(*
SPDX-FileCopyrightText: © 2026 Oleksandr Tiutyk <trofimich@gmail.com>
SPDX-License-Identifier: MIT
License: https://opensource.org/license/mit
*)

(*!
<summary>Wrapper for native exception codes. The manager's static instance is a shared borrowed view.</summary>
<description>
Dynamic instances/clones belong to DynamicMemoryManager and must not be deleted manually.
Framework propagation preserves the captured code, catch point and timestamps in a dynamic clone.
</description>
*)

//!<param name="_AutoDisposeRegistrar">Dynamic system exceptions share the manager-owned lifetime of other exceptions.</param>

{attribute 'enable_dynamic_creation'}	
{attribute 'no_explicit_call' := 'do not call this function block directly'} 


FUNCTION_BLOCK SystemException EXTENDS Object IMPLEMENTS IException
VAR
	{attribute 'hide'} 
	_ClassName : STRING := __POUNAME();

	{attribute 'hide'} 
	_ExceptionCode : __SYSTEM.ExceptionCode;
	_LocalTimestamp : LDATE_AND_TIME;
	_UtcTimestamp : LDATE_AND_TIME;
	{attribute 'hide'} 	
	_CatchPointNamespaceName : STRING;
	{attribute 'hide'} 
	_CatchPointPOUName : STRING;
	{attribute 'hide'} 
	_CatchPointPosition : STRING;
	
	{attribute 'hide'} 
	_UnspecifiedPOU : STRING(128);

	{attribute 'hide'} 
	_UnspecifiedPosition : STRING(32);

	
	_AutoDisposeRegistrar : AutoDisposeRegistrar(THIS^);
END_VAR

METHOD PRIVATE appendTimestampDescription
VAR_IN_OUT CONSTANT
	stringBuilder : WideStringBuilder;
END_VAR
VAR_INPUT
	timestampDisplayMode : TIMESTAMP_DISPLAY_MODE := TIMESTAMP_DISPLAY_MODE.HIDDEN;
	localTimestamp : LDATE_AND_TIME;	
	utcTimestamp : LDATE_AND_TIME;	
END_VAR
IF timestampDisplayMode = TIMESTAMP_DISPLAY_MODE.HIDDEN THEN
	RETURN;
END_IF

CASE timestampDisplayMode OF
	TIMESTAMP_DISPLAY_MODE.LOCAL:
		stringBuilder.Append(localTimestamp);
	
	TIMESTAMP_DISPLAY_MODE.UTC:
		stringBuilder.Append(utcTimestamp).AppendString("UTC");
END_CASE
END_METHOD

{attribute 'monitoring' := 'call'}
PROPERTY ClassName : REFERENCE TO STRING
GET
ClassName REF= _ClassName;
END_GET
END_PROPERTY

(*!
<summary>Clears the code: Empty becomes TRUE and GetMessage returns an empty string.</summary>
<description>
Resets captured timestamps; does not delete/unregister the instance. Catch-point storage is retained.
</description>
*)

METHOD Clear
_ExceptionCode := __SYSTEM.ExceptionCode.RTSEXCPT_NOEXCEPTION;
_LocalTimestamp := LongDateAndTimes.MIN_VALUE;
_UtcTimestamp := LongDateAndTimes.MIN_VALUE;
END_METHOD

(*!
<summary>Returns an auto-disposed copy of the code and catch point, borrowed until cleanup.</summary>
<description>
Captured timestamps are copied unchanged; cloning does not create a new occurrence time.
Allocation failure latches and raises fatal OUT_OF_MEMORY, without a heap exception.
</description>
*)

METHOD Clone : IObject
VAR
	exceptionClone : POINTER TO SystemException;
END_VAR
DynamicMemoryManager.RaiseIfAllocationFailed();
exceptionClone := __NEW(SystemException);

IF exceptionClone = 0 THEN
	DynamicMemoryManager.RaiseAllocationFailure();
	RETURN;
END_IF

exceptionClone^._ExceptionCode := _ExceptionCode;
exceptionClone^._CatchPointNamespaceName := _CatchPointNamespaceName;
exceptionClone^._CatchPointPOUName := _CatchPointPOUName;
exceptionClone^._CatchPointPosition := _CatchPointPosition;
exceptionClone^._LocalTimestamp := _LocalTimestamp;
exceptionClone^._UtcTimestamp := _UtcTimestamp;

Clone := exceptionClone^;
END_METHOD

(*!
<summary>Captures the time GetLastException observes the native exception, not the unavailable native throw time.</summary>
*)

METHOD INTERNAL Configure
VAR_IN_OUT CONSTANT
	exceptionCode : __SYSTEM.ExceptionCode;
	catchPointNamespaceName : STRING;
	catchPointPOUName : STRING;
	catchPointPosition : STRING;
END_VAR
_ExceptionCode := exceptionCode;
_CatchPointNamespaceName := catchPointNamespaceName;
_CatchPointPOUName := catchPointPOUName;
_CatchPointPosition := catchPointPosition;
_LocalTimestamp := System.SystemLocalDateTime;
_UtcTimestamp := System.SystemUtcDateTime;
END_METHOD

{attribute 'monitoring' := 'call'}
PROPERTY Empty : BOOL
GET
Empty := _ExceptionCode = __SYSTEM.ExceptionCode.RTSEXCPT_NOEXCEPTION;
END_GET
END_PROPERTY

{attribute 'monitoring' := 'call'}
PROPERTY FINAL ExceptionCode : __SYSTEM.ExceptionCode
GET
ExceptionCode := _ExceptionCode;
END_GET
END_PROPERTY

//!<param name="bInitRetains">if TRUE, the retain variables are initialized (warm start / cold start)</param>

//!<param name="bInCopyCode">if TRUE, the instance afterwards gets moved into the copy code (online change)</param>

METHOD FB_init : BOOL
VAR_INPUT
	
	bInitRetains	: BOOL;
	
	bInCopyCode	: BOOL;
END_VAR
_UnspecifiedPOU := Exceptions.UNSPECIFIED_SOURCE;
_UnspecifiedPosition := Exceptions.UNSPECIFIED_SOURCE;
END_METHOD

METHOD FINAL GetMessage : ERROR_MESSAGE
VAR_INPUT
	showSource : BOOL := FALSE;
	timestampDisplayMode : TIMESTAMP_DISPLAY_MODE := TIMESTAMP_DISPLAY_MODE.HIDDEN;
END_VAR
VAR
	stringBuilder : WideStringBuilder;
END_VAR
IF _ExceptionCode <> __SYSTEM.ExceptionCode.RTSEXCPT_NOEXCEPTION THEN
	stringBuilder
		.AppendString("System exception ")
		.AppendString255(TO_WSTRING(_ExceptionCode))
		.AppendString(" occured. Сaught in ")
		.AppendString255(TO_WSTRING(_CatchPointNamespaceName))
		.AppendString(".")
		.AppendString255(TO_WSTRING(_CatchPointPOUName))
		.AppendString(" at ")
		.AppendString255(TO_WSTRING(_CatchPointPosition));
			
	IF timestampDisplayMode <> TIMESTAMP_DISPLAY_MODE.HIDDEN THEN
		stringBuilder.AppendString(Exceptions.TIME_PREFIX);
		AppendTimestampDescription(stringBuilder, timestampDisplayMode, LocalTimestamp, UtcTimestamp);
	END_IF

	stringBuilder.AssignToString(GetMessage);
ELSE
	GetMessage := "";
END_IF
END_METHOD

METHOD FINAL GetRootException : IException
GetRootException := THIS^;
END_METHOD

METHOD FINAL GetSourceDescription : STRING(255)
GetSourceDescription := Exceptions.UNSPECIFIED_SOURCE;
END_METHOD

{attribute 'monitoring' := 'call'}
PROPERTY FINAL LocalTimestamp : LDATE_AND_TIME
GET
LocalTimestamp := _LocalTimestamp;
END_GET
END_PROPERTY

{attribute 'monitoring' := 'call'}
PROPERTY NamespaceName : REFERENCE TO STRING
GET
NamespaceName REF= CurrentNamespace.Name;
END_GET
END_PROPERTY

{attribute 'monitoring' := 'call'}
PROPERTY SelfSize : ULINT
GET
SelfSize := XSIZEOF(THIS^);
END_GET
END_PROPERTY

{attribute 'monitoring' := 'call'}
PROPERTY FINAL Severity : ERROR_SEVERITY
GET
Severity := ERROR_SEVERITY.CRITICAL;
END_GET
END_PROPERTY

{attribute 'monitoring' := 'call'}
PROPERTY FINAL SourceFullPOUName : REFERENCE TO STRING(128)
GET
SourceFullPOUName REF= _UnspecifiedPOU;
END_GET
END_PROPERTY

{attribute 'monitoring' := 'call'}
PROPERTY FINAL SourcePosition : REFERENCE TO STRING(32)
GET
SourcePosition REF= _UnspecifiedPosition;
END_GET
END_PROPERTY

METHOD ToError
VAR_IN_OUT CONSTANT
	targetError : ERROR;
END_VAR
VAR_INPUT
	severity : ERROR_SEVERITY;	
END_VAR
IF NOT __ISVALIDREF(targetError) THEN
	RETURN;
END_IF

targetError.Fill(
	severity,
	GetSourceDescription(),
	GetSourceDescription(),
	GetMessage(),
	GetMessage(),
	LocalTimestamp,
	UtcTimestamp
);
END_METHOD

{attribute 'monitoring' := 'call'}
PROPERTY FINAL UtcTimestamp : LDATE_AND_TIME
GET
UtcTimestamp := _UtcTimestamp;
END_GET
END_PROPERTY

END_FUNCTION_BLOCK

(* stored: Version 1.1.0.1
   POU SystemException: Id {003dda89-959c-4208-b47c-eab6a22da353}, SpecialFunc None
   Folder Service methods: Id {e40f07a0-bb69-43d2-9344-558beb521327}
   Method appendTimestampDescription: Id {dcf3179b-315e-43cb-bffb-a9cc08face8f}
   Property ClassName: Id {f6998750-94de-4b27-9017-ad7539ef8bae}
   Get Get: Id {cb7835e8-806f-4442-837f-895002f84c14}
   Method Clear: Id {dbd66dfc-fc8f-4256-a0f4-f74c9a16f7ea}
   Method Clone: Id {654edb60-f1ae-4e3d-854a-ef1384720f30}
   Method Configure: Id {297ea316-2fb7-4596-b05c-db0f46e37b1b}
   Property Empty: Id {038c5f5f-d26f-4e70-a390-6d5e8f198afd}
   Get Get: Id {60ffea73-58f0-48cd-a1b6-f69c50756f23}
   Property ExceptionCode: Id {98df4acc-7b54-406f-b517-a9c22c0f0d8e}
   Get Get: Id {90619a75-6b17-438b-a2b1-b465d62fd70b}
   Method FB_init: Id {9df7f179-6b56-448d-8f6f-07eac327896a}
   Method GetMessage: Id {a88a8b1a-9f6a-4c9d-9ec5-e6c280a6e922}
   Method GetRootException: Id {cfc4f0f7-35c9-4eb3-b854-bd2edbdcadfe}
   Method GetSourceDescription: Id {933b59e0-81e6-42d6-ba36-d2e00c47553a}
   Property LocalTimestamp: Id {243bf917-8856-414f-8657-d2ad403ee832}
   Get Get: Id {79d470da-f79a-4a33-bf4f-89aa38c370f7}
   Property NamespaceName: Id {ca510274-b070-4a45-bc4b-9eb8a5a40ec1}
   Get Get: Id {6c4acd0f-2e61-4a39-b5a8-d3f83794230d}
   Property SelfSize: Id {45a123fb-1e78-493d-ab14-ef856a5a55f6}
   Get Get: Id {adba8c9d-7fbf-47a5-ad28-a9aff99bf348}
   Property Severity: Id {5e42d487-fb84-4ef7-8167-9ccf2b832212}
   Get Get: Id {deb70a32-6e78-47a9-8646-53719a2a7ac5}
   Property SourceFullPOUName: Id {bb5b4681-7cbe-4420-8da3-3eab8d25b3a6}
   Get Get: Id {000c96a6-91dd-487f-a89a-7a0a528ae1fc}
   Property SourcePosition: Id {a0036bdf-f7b1-4700-90c9-8ba4e7777c8e}
   Get Get: Id {81eb6bc3-98ea-458a-b91b-7e4c86ab7dcc}
   Method ToError: Id {5bcd52e5-ca90-49d6-b86c-fe61de2dd705}
   Property UtcTimestamp: Id {b9a20ffe-1a2b-4d8b-a985-efb4f4570353}
   Get Get: Id {9ac21bad-7080-4914-9567-5b68982f14d9} *)
